FUNCTION_BLOCK SomeTestMultiPositions EXTENDS TcoDrivesBeckhoff.TcoMultiAxisPositionsRootContainer
VAR_INPUT
END_VAR
VAR_OUTPUT
END_VAR
VAR
	{attribute addProperty Name "<#Pick Position#>"}
	PickPosition:TcoDrivesBeckhoff.TcoMultiAxisMoveParam;
	{attribute addProperty Name "<#Place  Position#>"}
	PlacePosition:TcoDrivesBeckhoff.TcoMultiAxisMoveParam;

END_VAR

PROPERTY PUBLIC PickPos : REFERENCE TO TcoDrivesBeckhoff.TcoMultiAxisMoveParam;
GET
PickPos REF=PickPosition;
END_GET
END_PROPERTY

PROPERTY PUBLIC PlacePos : REFERENCE TO TcoDrivesBeckhoff.TcoMultiAxisMoveParam;
GET
PlacePos REF=PlacePosition;
END_GET
END_PROPERTY

END_FUNCTION_BLOCK

(* stored: Version 1.1.0.1, ProductVersion 3.1.4024.12
   POU SomeTestMultiPositions: Id {8273acfc-9b9e-0909-3854-4c84a6bea50d}, SpecialFunc None
   Property PickPos: Id {9afc3efe-977f-0cfa-2091-6b82330b36d7}
   Get Get: Id {54fd2e36-1768-0b24-3aaa-aa9fb0032d69}
   Property PlacePos: Id {48a58c59-a745-03be-305d-ea8c1e8e9873}
   Get Get: Id {51fcacf0-79b0-0952-0548-14f5f353edb9} *)
